ABB RobotStudio station: Trayectoria_1.rsstnx

Station Trayectoria_1 (saved by RobotStudio 23.4.10609.1)
Controller Controlador1
  mechanical unit ROB_1: IRB140_6_81_C_03, 6 joints, base frame (0, 0, 0) mm
Layout (positions relative to the parent item):
  - IRB140_6_81_C_03 [mechanism, from %ABB.RobotStudio.Models.IRB140%\IRB140_6_81_C_G_03.rslib] at (0, 0, 0) mm; joint values [0, 0, 0, 0, 0.5236, 0] (rad or m)
  - Porta_Marcador [mechanism] at (506.29, 0, 679.5) mm, rotated rx 180 ry 60 rz 180 deg
      TCP Punta at (90.51, 0, 143.01) mm, rotated rx 0 ry -45 rz 0 deg
      links: Support_RS_2
Attachment: Porta_Marcador is attached to IRB140_6_81_C_03 / Link6
Targets, tools, work objects and paths stored in the station, written as RAPID:
! task T_ROB1
MODULE CalibData
  PERS tooldata Punta:=[TRUE,[[90.50966799,0,143.009668],[0.923879533,0,-0.382683432,0]],[1,[0,0,1],[1,0,0,0],0,0,0]];
ENDMODULE

